FUNCTION_BLOCK FB_DB_CreateConnectionParams
VAR_INPUT
	bCreateNewConection					: BOOL;
END_VAR
VAR_OUTPUT
	bDBConnectionParamsCreated			: BOOL;
	bDBCreateConnectionError			: BOOL;
	nDBCreateConnectionError						: UDINT;
	sDBConnectionString					: STRING(255);
	nDBID								: UDINT;
END_VAR
VAR_IN_OUT
	stDBConfig										: ST_DB_Config;
END_VAR
VAR
	fbCreateConnection								: FB_DBConnectionAdd;
	ftrigCreationBusy				: F_TRIG;
	bConnectionAdded				: BOOL;
	test	: BOOL;
END_VAR

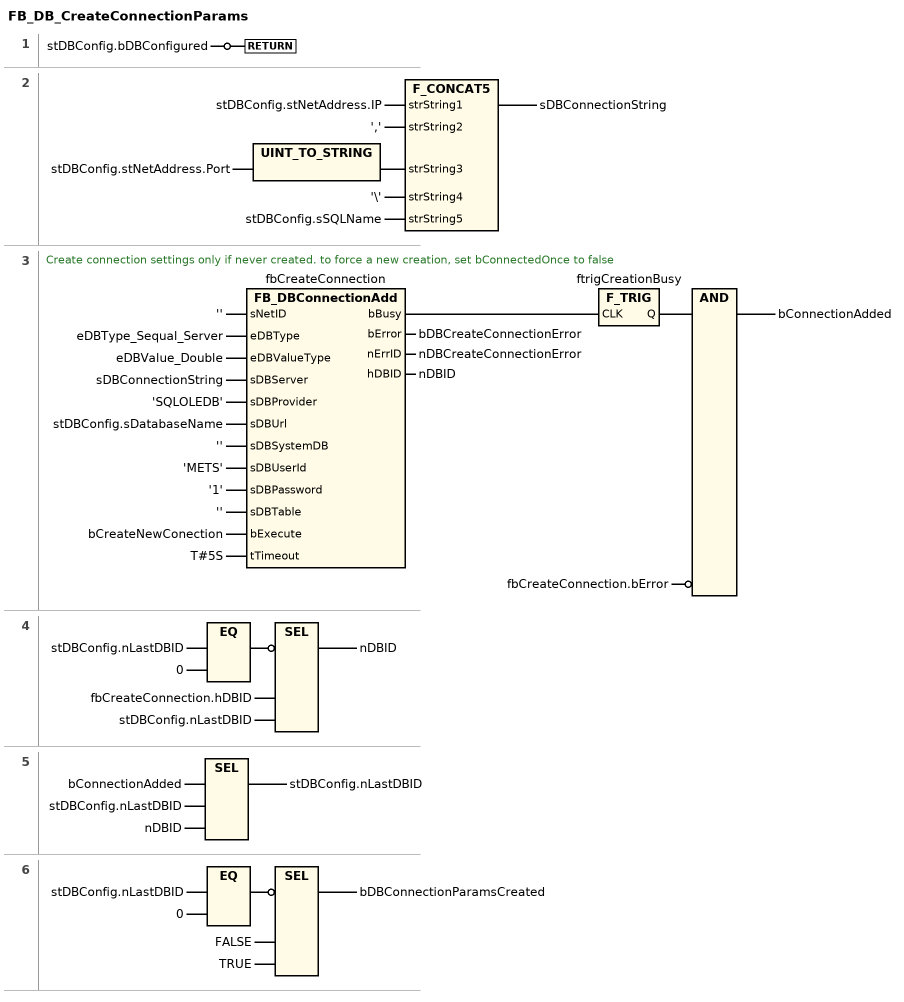
// NETWORK 1
IF NOT stDBConfig.bDBConfigured THEN RETURN; END_IF

// NETWORK 2
sDBConnectionString := F_CONCAT5(strString1 := stDBConfig.stNetAddress.IP, strString2 := ',', strString3 := UINT_TO_STRING(stDBConfig.stNetAddress.Port), strString4 := '\', strString5 := stDBConfig.sSQLName);

// NETWORK 3
// Create connection settings only if never created. to force a new creation, set bConnectedOnce to false
fbCreateConnection(
    sNetID := '',
    eDBType := eDBType_Sequal_Server,
    eDBValueType := eDBValue_Double,
    sDBServer := sDBConnectionString,
    sDBProvider := 'SQLOLEDB',
    sDBUrl := stDBConfig.sDatabaseName,
    sDBSystemDB := '',
    sDBUserId := 'METS',
    sDBPassword := '1',
    sDBTable := '',
    bExecute := bCreateNewConection,
    tTimeout := T#5S,
    bError => bDBCreateConnectionError,
    nErrID => nDBCreateConnectionError,
    hDBID => nDBID); // FB_DBConnectionAdd
ftrigCreationBusy(CLK := fbCreateConnection.bBusy); // F_TRIG
bConnectionAdded := ftrigCreationBusy.Q AND NOT fbCreateConnection.bError;

// NETWORK 4
nDBID := SEL(NOT (stDBConfig.nLastDBID = 0), fbCreateConnection.hDBID, stDBConfig.nLastDBID);

// NETWORK 5
stDBConfig.nLastDBID := SEL(bConnectionAdded, stDBConfig.nLastDBID, nDBID);

// NETWORK 6
bDBConnectionParamsCreated := SEL(NOT (stDBConfig.nLastDBID = 0), FALSE, TRUE);

END_FUNCTION_BLOCK

(* stored: Version 1.1.0.1, ProductVersion 3.1.4024.15
   POU FB_DB_CreateConnectionParams: Id {73853704-8766-454e-a30a-9f9a541b95d2}, SpecialFunc None *)
